// Tests exercise the public input/output and command contracts.
FUNCTION_BLOCK FB_AnalogInput_Test EXTENDS TcUnit.FB_TestSuite
VAR CONSTANT
    TOL : REAL := 1E-3;
END_VAR

InitialStatusPublishesDefaults();
LinearScalingMapsEndpointsAndMidpoint();
RawBypassSkipsClampAndScaling();
ClampLowReportsAndHoldsAtRawMin();
ClampHighReportsAndHoldsAtRawMax();
ClampPromotesGoodQualityToClamped();
ClampAsFaultRaisesClampLow();
ClampAsFaultRaisesClampHigh();
BadConfigRaisesFaultOnFirstScan();
BadQualityHoldsLastRawReading();
InputTypeRealReadsRealMemberOfUnion();
QualityTagPropagatesToStatus();

METHOD InitialStatusPublishesDefaults
VAR
    fb : TcForge.FB_AnalogInput;
END_VAR
TEST('InitialStatusPublishesDefaults');

// Default cfg: INT terminal, raw 0..32767 -> EU 0..100, no filter,
// clamp-as-fault disabled. The application must explicitly label the unit.
// With inRaw zero-initialised the first cycle reports a clean 0 and no fault.
fb(inpQuality := TcForge.E_IO_Quality.GOOD);

AssertTrue(
    Condition := fb.sts.unit = TcForge.E_Unit.UNSPECIFIED,
    Message   := 'An unconfigured channel must not claim a physical unit');

AssertTrue(
    Condition := ABS(fb.sts.value) < TOL,
    Message   := 'Fresh instance must publish value = 0 for a raw input of 0');
AssertTrue(
    Condition := ABS(fb.sts.rawReal) < TOL,
    Message   := 'Fresh instance must publish rawReal = 0');
AssertFalse(
    Condition := fb.sts.clampActive,
    Message   := 'Raw 0 is inside [0, 32767] so clampActive must be FALSE');
AssertFalse(
    Condition := fb.sts.header.faulted,
    Message   := 'Fresh instance must not be faulted');

TEST_FINISHED();
END_METHOD

METHOD LinearScalingMapsEndpointsAndMidpoint
VAR
    fb : TcForge.FB_AnalogInput;
END_VAR
TEST('LinearScalingMapsEndpointsAndMidpoint');

// Default cfg: raw 0..32767 -> EU 0..100. Verify the two endpoints and
// the midpoint land where the linear recurrence says they should.
//
//     value = euMin + (raw - rawMin)
//                           * (euMax - euMin)
//                           / (rawMax - rawMin)

fb.inRaw.nInt := 0;
fb(inpQuality := TcForge.E_IO_Quality.GOOD);
AssertTrue(
    Condition := ABS(fb.sts.value - 0.0) < TOL,
    Message   := 'Raw = rawMin must map to euMin (0 %)');

fb.inRaw.nInt := 32767;
fb(inpQuality := TcForge.E_IO_Quality.GOOD);
AssertTrue(
    Condition := ABS(fb.sts.value - 100.0) < TOL,
    Message   := 'Raw = rawMax must map to euMax (100 %)');

fb.inRaw.nInt := 16384;
fb(inpQuality := TcForge.E_IO_Quality.GOOD);
AssertTrue(
    Condition := ABS(fb.sts.value - 50.0015) < 0.01,
    Message   := 'Raw ~ midpoint must map to EU ~ 50 %');

TEST_FINISHED();
END_METHOD

METHOD RawBypassSkipsClampAndScaling
VAR
    fb : TcForge.FB_AnalogInput;
END_VAR
TEST('RawBypassSkipsClampAndScaling');

// useRawValue = TRUE publishes the raw REAL directly and suppresses
// the clamp flags even when the raw value is outside the scaling range.
fb.cfg.useRawValue := TRUE;
fb.inRaw.nInt := 30000;
fb(inpQuality := TcForge.E_IO_Quality.GOOD);

AssertTrue(
    Condition := ABS(fb.sts.value - fb.sts.rawReal) < TOL,
    Message   := 'With useRawValue = TRUE, value must equal rawReal');
AssertFalse(
    Condition := fb.sts.clampedLow,
    Message   := 'Raw bypass must not flag clampedLow');
AssertFalse(
    Condition := fb.sts.clampedHigh,
    Message   := 'Raw bypass must not flag clampedHigh');
AssertFalse(
    Condition := fb.sts.clampActive,
    Message   := 'Raw bypass must not flag clampActive');

TEST_FINISHED();
END_METHOD

METHOD ClampLowReportsAndHoldsAtRawMin
VAR
    fb : TcForge.FB_AnalogInput;
END_VAR
TEST('ClampLowReportsAndHoldsAtRawMin');

// Drive the raw INT below rawMin. The clamp must flag clampedLow
// and pin the scaled value at euMin.
fb.inRaw.nInt := -500;
fb(inpQuality := TcForge.E_IO_Quality.GOOD);

AssertTrue(
    Condition := fb.sts.clampedLow,
    Message   := 'Raw below rawMin must set clampedLow');
AssertTrue(
    Condition := fb.sts.clampActive,
    Message   := 'clampActive must be TRUE whenever either clamp direction is active');
AssertTrue(
    Condition := ABS(fb.sts.value - 0.0) < TOL,
    Message   := 'Clamped-low output must pin to euMin (0 %)');
AssertFalse(
    Condition := fb.sts.header.faulted,
    Message   := 'clampAsFault = FALSE by default; clamp alone must not fault the device');

TEST_FINISHED();
END_METHOD

METHOD ClampHighReportsAndHoldsAtRawMax
VAR
    fb : TcForge.FB_AnalogInput;
END_VAR
TEST('ClampHighReportsAndHoldsAtRawMax');

// Use REAL input so we can inject a raw that is clearly above rawMax
// (INT saturates at 32767; REAL doesn't).
fb.cfg.inputType := __SYSTEM.TYPE_CLASS.TYPE_REAL;
fb.inRaw.fReal := 40000.0;
fb(inpQuality := TcForge.E_IO_Quality.GOOD);

AssertTrue(
    Condition := fb.sts.clampedHigh,
    Message   := 'Raw above rawMax must set clampedHigh');
AssertTrue(
    Condition := fb.sts.clampActive,
    Message   := 'clampActive must be TRUE when clampedHigh is set');
AssertTrue(
    Condition := ABS(fb.sts.value - 100.0) < TOL,
    Message   := 'Clamped-high output must pin to euMax (100 %)');

TEST_FINISHED();
END_METHOD

METHOD ClampPromotesGoodQualityToClamped
VAR
    fb : TcForge.FB_AnalogInput;
END_VAR
TEST('ClampPromotesGoodQualityToClamped');

// When the raw input is clamping *and* inpQuality = GOOD, the FB must
// promote quality to CLAMPED to signal "reading is legal but pinned".
fb.inRaw.nInt := -1;
fb(inpQuality := TcForge.E_IO_Quality.GOOD);

AssertTrue(
    Condition := fb.sts.clampActive,
    Message   := 'Precondition: clampActive must be TRUE');
AssertEquals_DINT(
    Expected := TO_DINT(TcForge.E_IO_Quality.CLAMPED),
    Actual   := TO_DINT(fb.sts.quality),
    Message  := 'GOOD quality must be promoted to CLAMPED while clamping');

TEST_FINISHED();
END_METHOD

METHOD ClampAsFaultRaisesClampLow
VAR
    fb : TcForge.FB_AnalogInput;
END_VAR
TEST('ClampAsFaultRaisesClampLow');

fb.cfg.clampAsFault := TRUE;
fb.inRaw.nInt := -10;
fb(inpQuality := TcForge.E_IO_Quality.GOOD);

AssertTrue(
    Condition := fb.sts.header.faulted,
    Message   := 'clampAsFault + raw below RawMin must fault the device');
AssertEquals_DINT(
    Expected := TcForge.E_AnalogInput_Fault.ClampLow,
    Actual   := fb.sts.header.faultCode,
    Message  := 'Fault code must be ClampLow');

TEST_FINISHED();
END_METHOD

METHOD ClampAsFaultRaisesClampHigh
VAR
    fb : TcForge.FB_AnalogInput;
END_VAR
TEST('ClampAsFaultRaisesClampHigh');

fb.cfg.clampAsFault := TRUE;
fb.cfg.inputType    := __SYSTEM.TYPE_CLASS.TYPE_REAL;
fb.inRaw.fReal := 50000.0;
fb(inpQuality := TcForge.E_IO_Quality.GOOD);

AssertTrue(
    Condition := fb.sts.header.faulted,
    Message   := 'clampAsFault + raw above RawMax must fault the device');
AssertEquals_DINT(
    Expected := TcForge.E_AnalogInput_Fault.ClampHigh,
    Actual   := fb.sts.header.faultCode,
    Message  := 'Fault code must be ClampHigh');

TEST_FINISHED();
END_METHOD

METHOD BadConfigRaisesFaultOnFirstScan
VAR
    fb : TcForge.FB_AnalogInput;
END_VAR
TEST('BadConfigRaisesFaultOnFirstScan');

// BadConfig check runs once on the first scan. Set rawMin >= rawMax
// BEFORE the first cyclic call so the validation can latch _configBad.
fb.cfg.rawMin := 100.0;
fb.cfg.rawMax := 100.0;
fb(inpQuality := TcForge.E_IO_Quality.GOOD);

AssertTrue(
    Condition := fb.sts.header.faulted,
    Message   := 'rawMin >= rawMax must fault the device as BadConfig');
AssertEquals_DINT(
    Expected := TcForge.E_AnalogInput_Fault.BadConfig,
    Actual   := fb.sts.header.faultCode,
    Message  := 'Fault code must be BadConfig');

TEST_FINISHED();
END_METHOD

METHOD BadQualityHoldsLastRawReading
VAR
    fb          : TcForge.FB_AnalogInput;
    snapshotRaw : REAL;
END_VAR
TEST('BadQualityHoldsLastRawReading');

// Establish a good reading first.
fb.inRaw.nInt := 10000;
fb(inpQuality := TcForge.E_IO_Quality.GOOD);
snapshotRaw := fb.sts.rawReal;

// Flip quality to BAD and change the raw wire. The FB must discard the
// fresh value and hold the last-known-good raw reading.
fb.inRaw.nInt := 25000;
fb(inpQuality := TcForge.E_IO_Quality.BAD);

AssertTrue(
    Condition := ABS(fb.sts.rawReal - snapshotRaw) < TOL,
    Message   := 'BAD quality must hold rawReal at the last-known-good value');

TEST_FINISHED();
END_METHOD

METHOD InputTypeRealReadsRealMemberOfUnion
VAR
    fb : TcForge.FB_AnalogInput;
END_VAR
TEST('InputTypeRealReadsRealMemberOfUnion');

// Select the REAL UNION member and reconfigure scaling so raw == EU,
// then confirm the FB reads the REAL alias rather than some other
// reinterpretation of the same bytes.
fb.cfg.inputType := __SYSTEM.TYPE_CLASS.TYPE_REAL;
fb.cfg.rawMin    := 0.0;
fb.cfg.rawMax    := 100.0;
fb.cfg.euMin     := 0.0;
fb.cfg.euMax     := 100.0;

fb.inRaw.fReal := 42.5;
fb(inpQuality := TcForge.E_IO_Quality.GOOD);

AssertTrue(
    Condition := ABS(fb.sts.rawReal - 42.5) < TOL,
    Message   := 'TYPE_REAL must read inRaw.fReal directly into rawReal');
AssertTrue(
    Condition := ABS(fb.sts.value - 42.5) < TOL,
    Message   := 'Identity scaling must leave value equal to the raw REAL input');

TEST_FINISHED();
END_METHOD

METHOD QualityTagPropagatesToStatus
VAR
    fb : TcForge.FB_AnalogInput;
END_VAR
TEST('QualityTagPropagatesToStatus');

// The FB must echo inpQuality into sts.quality each cycle (subject to
// the clamp promotion covered by ClampPromotesGoodQualityToClamped).
fb.inRaw.nInt := 10000;
fb(inpQuality := TcForge.E_IO_Quality.GOOD);
AssertEquals_DINT(
    Expected := TO_DINT(TcForge.E_IO_Quality.GOOD),
    Actual   := TO_DINT(fb.sts.quality),
    Message  := 'quality must mirror inpQuality = GOOD when not clamping');

fb(inpQuality := TcForge.E_IO_Quality.UNKNOWN);
AssertEquals_DINT(
    Expected := TO_DINT(TcForge.E_IO_Quality.UNKNOWN),
    Actual   := TO_DINT(fb.sts.quality),
    Message  := 'quality must mirror inpQuality = UNKNOWN');

fb(inpQuality := TcForge.E_IO_Quality.BAD);
AssertEquals_DINT(
    Expected := TO_DINT(TcForge.E_IO_Quality.BAD),
    Actual   := TO_DINT(fb.sts.quality),
    Message  := 'quality must mirror inpQuality = BAD');

TEST_FINISHED();
END_METHOD

END_FUNCTION_BLOCK

(* stored: Version 1.1.0.1, ProductVersion 3.1.4026.12
   POU FB_AnalogInput_Test: Id {b1c2d3e4-f5a6-7890-abcd-000000000e00}, SpecialFunc None
   Method InitialStatusPublishesDefaults: Id {b1c2d3e4-f5a6-7890-abcd-000000000e01}
   Method LinearScalingMapsEndpointsAndMidpoint: Id {b1c2d3e4-f5a6-7890-abcd-000000000e02}
   Method RawBypassSkipsClampAndScaling: Id {b1c2d3e4-f5a6-7890-abcd-000000000e03}
   Method ClampLowReportsAndHoldsAtRawMin: Id {b1c2d3e4-f5a6-7890-abcd-000000000e04}
   Method ClampHighReportsAndHoldsAtRawMax: Id {b1c2d3e4-f5a6-7890-abcd-000000000e05}
   Method ClampPromotesGoodQualityToClamped: Id {b1c2d3e4-f5a6-7890-abcd-000000000e06}
   Method ClampAsFaultRaisesClampLow: Id {b1c2d3e4-f5a6-7890-abcd-000000000e07}
   Method ClampAsFaultRaisesClampHigh: Id {b1c2d3e4-f5a6-7890-abcd-000000000e08}
   Method BadConfigRaisesFaultOnFirstScan: Id {b1c2d3e4-f5a6-7890-abcd-000000000e09}
   Method BadQualityHoldsLastRawReading: Id {b1c2d3e4-f5a6-7890-abcd-000000000e0a}
   Method InputTypeRealReadsRealMemberOfUnion: Id {b1c2d3e4-f5a6-7890-abcd-000000000e0b}
   Method QualityTagPropagatesToStatus: Id {b1c2d3e4-f5a6-7890-abcd-000000000e0c} *)
